
// ===== library: MasterCopy "SeachArray[FC001]" =====

FUNCTION "SeachArray[FC001]" : Void   // FC4, LAD
{ S7_Optimized_Access := 'TRUE' }
VERSION : 0.1
   VAR_INPUT
      StartSearch : Bool;
      Search : DInt;
      UserArray : Array[0..99] of Struct
         RFID : DInt;
         "Name" : String;
         ClockNumber : Int;
         AccessLevel : Int;
      END_STRUCT;
      Reset : Bool;
   END_VAR
   VAR_OUTPUT
      MatchFound : Bool;
      NoMatchFound : Bool;
      MatchIndex : Int;
      EmptyIndex : Int;
      ArrayFull : Bool;
      Done : Bool;
   END_VAR
   VAR_TEMP
      Index : Int;
      Match : Bool;
      NoMatch : Bool;
   END_VAR
   VAR CONSTANT
      Null : String;
   END_VAR
   VAR_TEMP   // added for the SCL form of the ladder/FBD networks
      _w1 : Bool;
      _w2 : Bool;
   END_VAR
BEGIN

REGION Network 1: Search For Matching RFID
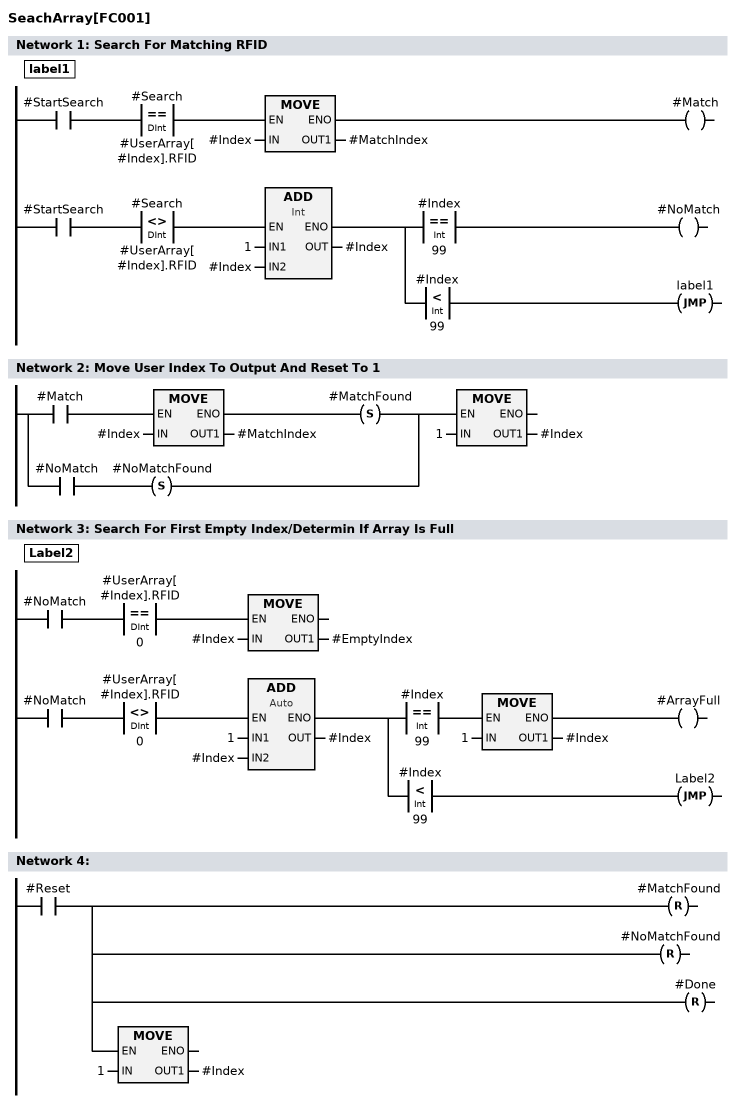
   Label( label1 )
   RUNG wire#powerrail
      Contact( #StartSearch )
      { S7_Templates := "SrcType := DInt" } EQ_Contact(in1 := #Search, in2 := #UserArray[#Index].RFID)
      Move(in := #Index, out1 => #MatchIndex)
      Coil( #Match )
   END_RUNG
   RUNG wire#powerrail
      Contact( #StartSearch )
      { S7_Templates := "SrcType := DInt" } NE_Contact(in1 := #Search, in2 := #UserArray[#Index].RFID)
      { S7_Templates := "SrcType := Int" } Add(in1 := 1, in2 := #Index, out => #Index)
      wire#w1
      { S7_Templates := "SrcType := Int" } EQ_Contact(in1 := #Index, in2 := 99)
      Coil( #NoMatch )
   END_RUNG
   RUNG wire#w1
      { S7_Templates := "SrcType := Int" } LT_Contact(in1 := #Index, in2 := 99)
      JumpCoil( label1 )
   END_RUNG
   // the same network as SCL:
   label1:
   #_w1 := #StartSearch AND (#Search = #UserArray[#Index].RFID);
   IF #_w1 THEN #MatchIndex := #Index; END_IF;
   #Match := #_w1;
   #_w2 := #StartSearch AND (#Search <> #UserArray[#Index].RFID);
   IF #_w2 THEN #Index := 1 + #Index; END_IF;
   #NoMatch := #_w2 AND (#Index = 99);
   IF #_w2 AND (#Index < 99) THEN GOTO label1; END_IF;
END_REGION

REGION Network 2: Move User Index To Output And Reset To 1
   RUNG wire#powerrail
      Contact( #Match )
      Move(in := #Index, out1 => #MatchIndex)
      S_Coil( #MatchFound )
      wire#w1
      Move(in := 1, out1 => #Index)
   END_RUNG
   RUNG wire#powerrail
      Contact( #NoMatch )
      S_Coil( #NoMatchFound )
   END_RUNG wire#w1
   // the same network as SCL:
   IF #Match THEN
       #MatchIndex := #Index;
       #MatchFound := TRUE;
   END_IF;
   IF #NoMatch THEN #NoMatchFound := TRUE; END_IF;
   IF #Match OR #NoMatch THEN #Index := 1; END_IF;
END_REGION

REGION Network 3: Search For First Empty Index/Determin If Array Is Full
   Label( Label2 )
   RUNG wire#powerrail
      Contact( #NoMatch )
      { S7_Templates := "SrcType := DInt" } EQ_Contact(in1 := #UserArray[#Index].RFID, in2 := 0)
      Move(in := #Index, out1 => #EmptyIndex)
   END_RUNG
   RUNG wire#powerrail
      Contact( #NoMatch )
      { S7_Templates := "SrcType := DInt" } NE_Contact(in1 := #UserArray[#Index].RFID, in2 := 0)
      Add(in1 := 1, in2 := #Index, out => #Index)
      wire#w1
      { S7_Templates := "SrcType := Int" } EQ_Contact(in1 := #Index, in2 := 99)
      Move(in := 1, out1 => #Index)
      Coil( #ArrayFull )
   END_RUNG
   RUNG wire#w1
      { S7_Templates := "SrcType := Int" } LT_Contact(in1 := #Index, in2 := 99)
      JumpCoil( Label2 )
   END_RUNG
   // the same network as SCL:
   Label2:
   IF #NoMatch AND (#UserArray[#Index].RFID = 0) THEN #EmptyIndex := #Index; END_IF;
   #_w1 := #NoMatch AND (#UserArray[#Index].RFID <> 0);
   IF #_w1 THEN #Index := 1 + #Index; END_IF;
   #_w2 := #_w1 AND (#Index = 99);
   IF #_w2 THEN #Index := 1; END_IF;
   #ArrayFull := #_w2;
   IF #_w1 AND (#Index < 99) THEN GOTO Label2; END_IF;
END_REGION

REGION Network 4
   RUNG wire#powerrail
      Contact( #Reset )
      wire#w1
      R_Coil( #MatchFound )
   END_RUNG
   RUNG wire#w1
      R_Coil( #NoMatchFound )
   END_RUNG
   RUNG wire#w1
      R_Coil( #Done )
   END_RUNG
   RUNG wire#w1
      Move(in := 1, out1 => #Index)
   END_RUNG
   // the same network as SCL:
   IF #Reset THEN
       #MatchFound := FALSE;
       #NoMatchFound := FALSE;
       #Done := FALSE;
       #Index := 1;
   END_IF;
END_REGION
END_FUNCTION

// ===== library: MasterCopy "LabelPrintEthernet" =====

FUNCTION "BuildLabel" : Void   // FC1, LAD
{ S7_Optimized_Access := 'TRUE' }
VERSION : 0.1
   VAR_INPUT
      REQ : Bool;
      PartNumber : String;
      PartDisctription : String;
      SerialNumber : Int;
      IPAddress1 : Byte;
      IPAddress2 : Byte;
      IPAddress3 : Byte;
      IPAddress4 : Byte;
      Port : UInt;
   END_VAR
   VAR_OUTPUT
      FinalLabel : String;
   END_VAR
   VAR_TEMP
      LabelDateTime : DTL;
      YearString : String;
      MonthString : String;
      DayString : String;
      HourString : String;
      MinuteString : String;
      SecondString : String;
      DateTimeString : String;
      AssembleLabel : String;
      SerialNumberString : String;
      BarcodeString : String;
      SerialNumberStringTemp : String;
      PrintData : String;
   END_VAR
   VAR CONSTANT
      FormatStart : String := '^XA';
      FormatLine1 : String := '^FS^A0N15,35^FO300,40^FD';
      FormatLine2 : String := '^FS^A0N20,20^FO300,80^FD';
      FormatLine3 : String := '^FS^A0N20,20^FO300,120^FD';
      FormatBarcode1 : String := '^FS^BXN,.05,200,^FO150,70^FD';
      FormatBarcode2 : String := '^FS^BXN,.04,200,^FO500,120^FD';
      FormatEnd : String := '^FS^XZ';
   END_VAR
BEGIN

REGION Network 1
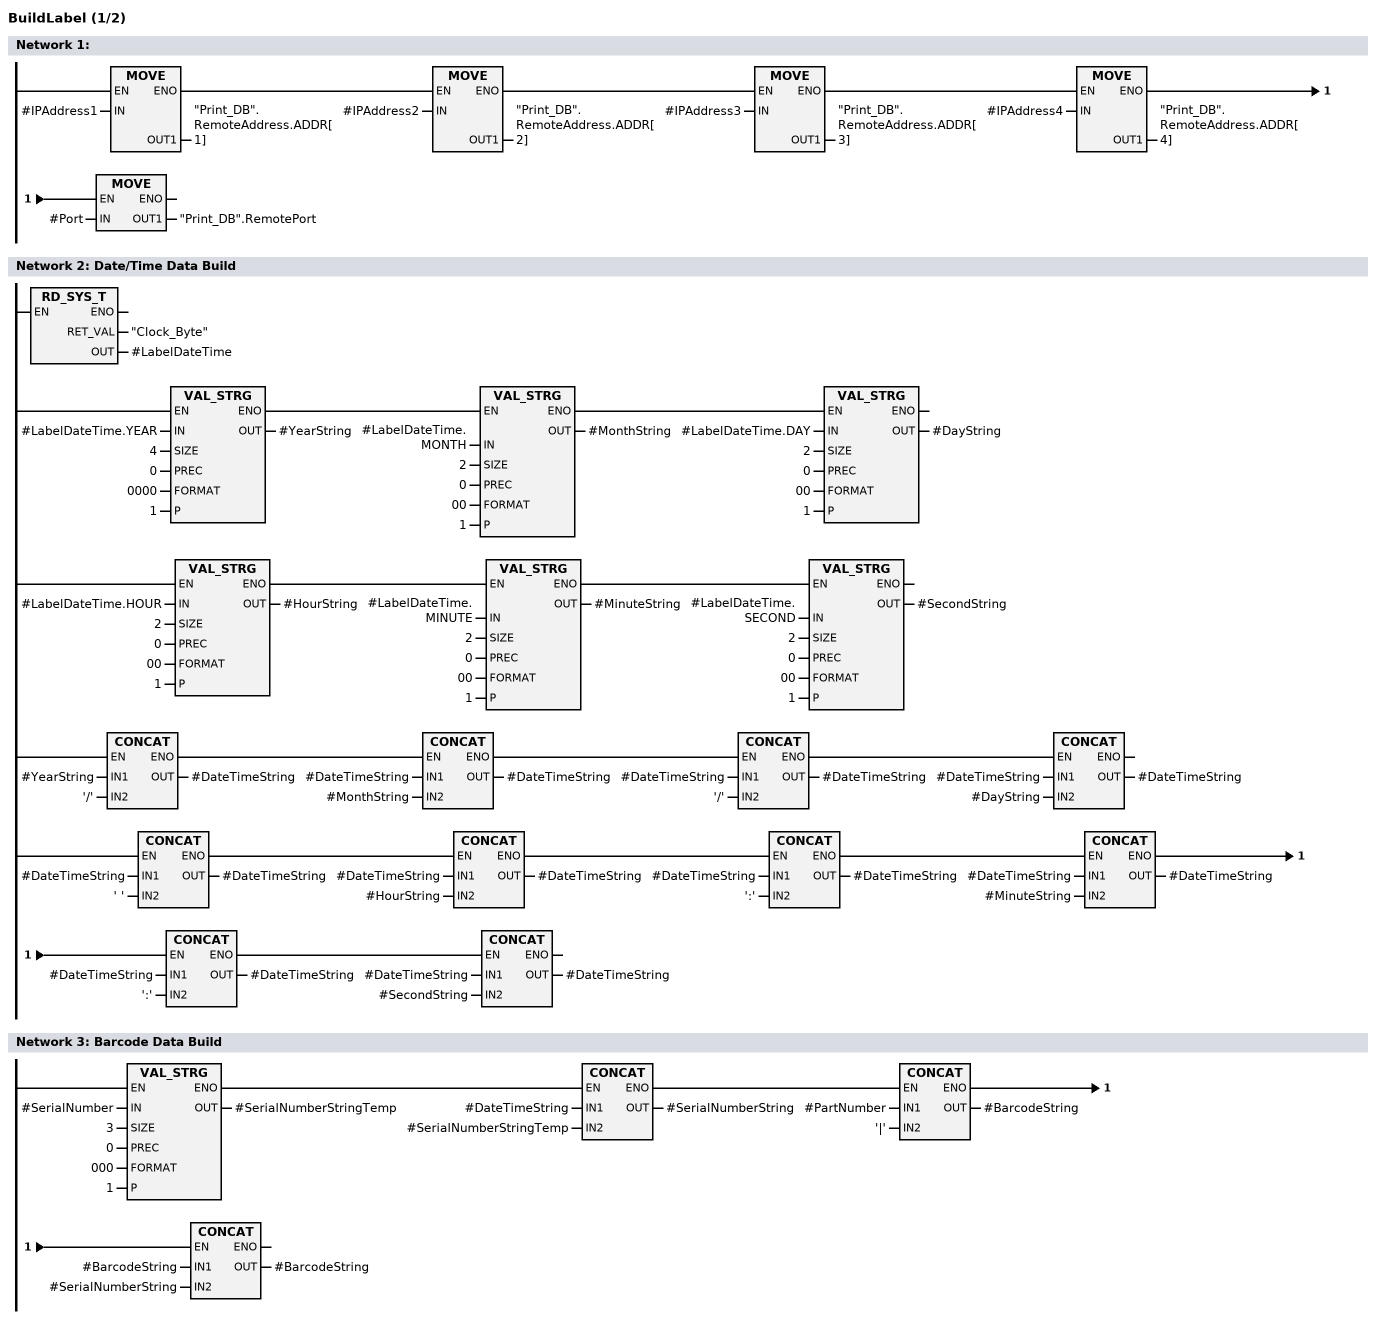
   RUNG wire#powerrail
      Move(in := #IPAddress1, out1 => "Print_DB".RemoteAddress.ADDR[1])
      Move(in := #IPAddress2, out1 => "Print_DB".RemoteAddress.ADDR[2])
      Move(in := #IPAddress3, out1 => "Print_DB".RemoteAddress.ADDR[3])
      Move(in := #IPAddress4, out1 => "Print_DB".RemoteAddress.ADDR[4])
      Move(in := #Port, out1 => "Print_DB".RemotePort)
   END_RUNG
   // the same network as SCL:
   "Print_DB".RemoteAddress.ADDR[1] := #IPAddress1;
   "Print_DB".RemoteAddress.ADDR[2] := #IPAddress2;
   "Print_DB".RemoteAddress.ADDR[3] := #IPAddress3;
   "Print_DB".RemoteAddress.ADDR[4] := #IPAddress4;
   "Print_DB".RemotePort := #Port;
END_REGION

REGION Network 2: Date/Time Data Build
   // ENO of a box is taken as its EN; it also drops when the box reports an error
   "Clock_Byte" := RD_SYS_T(OUT => #LabelDateTime);
   VAL_STRG(IN := #LabelDateTime.YEAR, SIZE := 4, PREC := 0, FORMAT := 0000, P := 1, OUT => #YearString);
   VAL_STRG(IN := #LabelDateTime.MONTH, SIZE := 2, PREC := 0, FORMAT := 00, P := 1, OUT => #MonthString);
   VAL_STRG(IN := #LabelDateTime.DAY, SIZE := 2, PREC := 0, FORMAT := 00, P := 1, OUT => #DayString);
   VAL_STRG(IN := #LabelDateTime.HOUR, SIZE := 2, PREC := 0, FORMAT := 00, P := 1, OUT => #HourString);
   VAL_STRG(IN := #LabelDateTime.MINUTE, SIZE := 2, PREC := 0, FORMAT := 00, P := 1, OUT => #MinuteString);
   VAL_STRG(IN := #LabelDateTime.SECOND, SIZE := 2, PREC := 0, FORMAT := 00, P := 1, OUT => #SecondString);
   #DateTimeString := CONCAT(IN1 := #YearString, IN2 := '/');
   #DateTimeString := CONCAT(IN1 := #DateTimeString, IN2 := #MonthString);
   #DateTimeString := CONCAT(IN1 := #DateTimeString, IN2 := '/');
   #DateTimeString := CONCAT(IN1 := #DateTimeString, IN2 := #DayString);
   #DateTimeString := CONCAT(IN1 := #DateTimeString, IN2 := ' ');
   #DateTimeString := CONCAT(IN1 := #DateTimeString, IN2 := #HourString);
   #DateTimeString := CONCAT(IN1 := #DateTimeString, IN2 := ':');
   #DateTimeString := CONCAT(IN1 := #DateTimeString, IN2 := #MinuteString);
   #DateTimeString := CONCAT(IN1 := #DateTimeString, IN2 := ':');
   #DateTimeString := CONCAT(IN1 := #DateTimeString, IN2 := #SecondString);
END_REGION

REGION Network 3: Barcode Data Build
   // ENO of a box is taken as its EN; it also drops when the box reports an error
   VAL_STRG(IN := #SerialNumber, SIZE := 3, PREC := 0, FORMAT := 000, P := 1, OUT => #SerialNumberStringTemp);
   #SerialNumberString := CONCAT(IN1 := #DateTimeString, IN2 := #SerialNumberStringTemp);
   #BarcodeString := CONCAT(IN1 := #PartNumber, IN2 := '|');
   #BarcodeString := CONCAT(IN1 := #BarcodeString, IN2 := #SerialNumberString);
END_REGION

REGION Network 4: Label Data Build
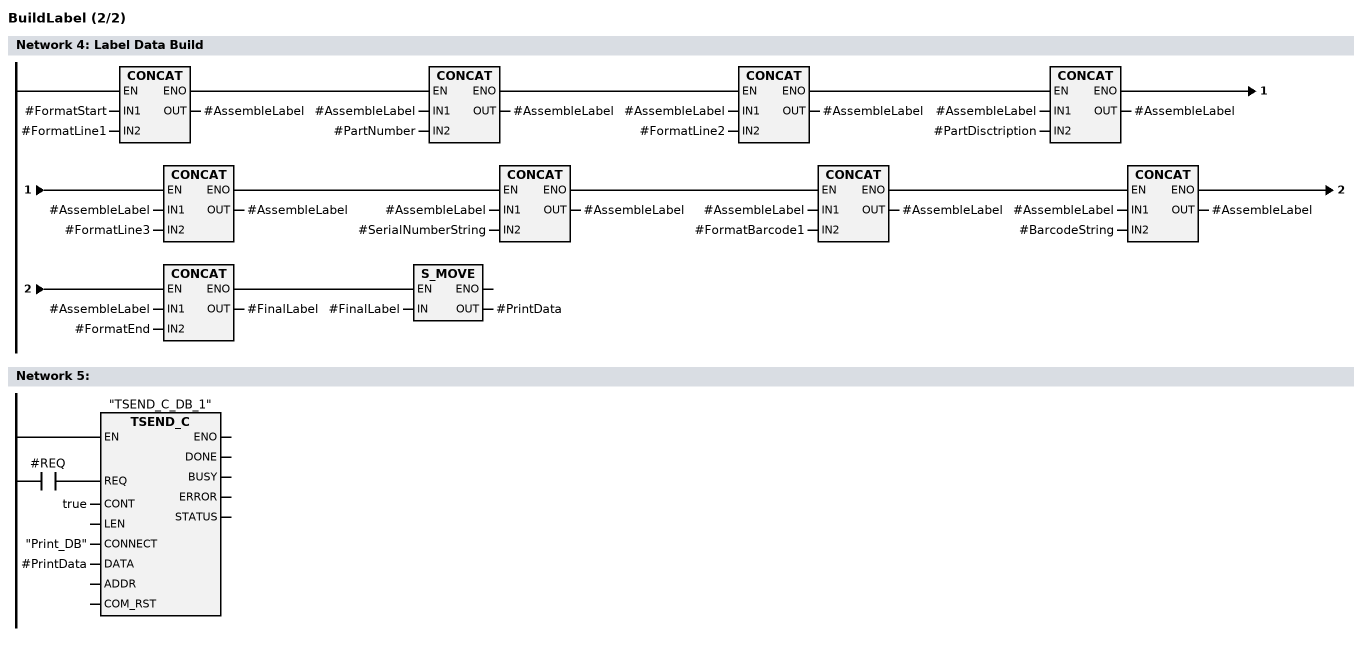
   #AssembleLabel := CONCAT(IN1 := #FormatStart, IN2 := #FormatLine1);
   #AssembleLabel := CONCAT(IN1 := #AssembleLabel, IN2 := #PartNumber);
   #AssembleLabel := CONCAT(IN1 := #AssembleLabel, IN2 := #FormatLine2);
   #AssembleLabel := CONCAT(IN1 := #AssembleLabel, IN2 := #PartDisctription);
   #AssembleLabel := CONCAT(IN1 := #AssembleLabel, IN2 := #FormatLine3);
   #AssembleLabel := CONCAT(IN1 := #AssembleLabel, IN2 := #SerialNumberString);
   #AssembleLabel := CONCAT(IN1 := #AssembleLabel, IN2 := #FormatBarcode1);
   #AssembleLabel := CONCAT(IN1 := #AssembleLabel, IN2 := #BarcodeString);
   #FinalLabel := CONCAT(IN1 := #AssembleLabel, IN2 := #FormatEnd);
   #PrintData := #FinalLabel;
END_REGION

REGION Network 5
   "TSEND_C_DB_1"(REQ := #REQ, CONT := true, CONNECT := "Print_DB", DATA := #PrintData);   // TSEND_C
END_REGION
END_FUNCTION

// ===== library: MasterCopy "Banner_IOLink_K50L" =====

FUNCTION "Banner_IOLink_K50L" : Void   // FC6, LAD
{ S7_Optimized_Access := 'TRUE' }
VERSION : 0.1
   VAR_INPUT
      IN : Bool;
      "Color 1" : Int;
      "Color 1 Intensity" : Int;
      "Color 2" : Int;
      "Color 2 Intensity" : Int;
      "Animation Type" : Int;
      "Rotation Direction" : Bool;
      "Flash Rate" : Int;
   END_VAR
BEGIN

REGION Network 1
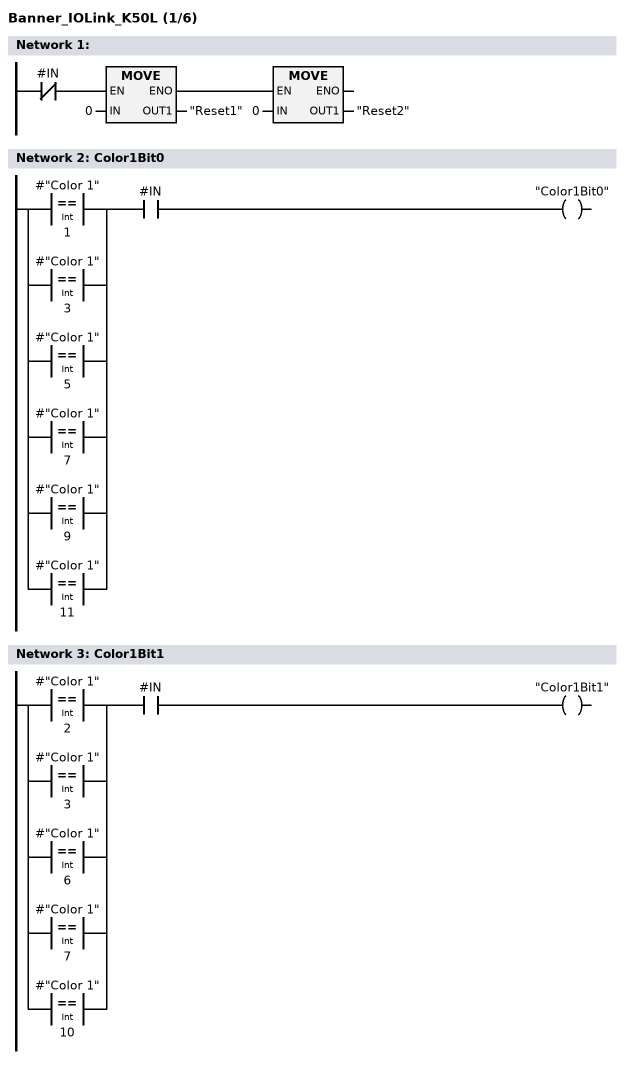
   RUNG wire#powerrail
      I_Contact( #IN )
      Move(in := 0, out1 => "Reset1")
      Move(in := 0, out1 => "Reset2")
   END_RUNG
   // the same network as SCL:
   IF NOT #IN THEN
       "Reset1" := 0;
       "Reset2" := 0;
   END_IF;
END_REGION

REGION Network 2: Color1Bit0
   RUNG wire#powerrail
      { S7_Templates := "SrcType := Int" } EQ_Contact(in1 := #"Color 1", in2 := 1)
      wire#w1
      Contact( #IN )
      Coil( "Color1Bit0" )
   END_RUNG
   RUNG wire#powerrail
      { S7_Templates := "SrcType := Int" } EQ_Contact(in1 := #"Color 1", in2 := 3)
   END_RUNG wire#w1
   RUNG wire#powerrail
      { S7_Templates := "SrcType := Int" } EQ_Contact(in1 := #"Color 1", in2 := 5)
   END_RUNG wire#w1
   RUNG wire#powerrail
      { S7_Templates := "SrcType := Int" } EQ_Contact(in1 := #"Color 1", in2 := 7)
   END_RUNG wire#w1
   RUNG wire#powerrail
      { S7_Templates := "SrcType := Int" } EQ_Contact(in1 := #"Color 1", in2 := 9)
   END_RUNG wire#w1
   RUNG wire#powerrail
      { S7_Templates := "SrcType := Int" } EQ_Contact(in1 := #"Color 1", in2 := 11)
   END_RUNG wire#w1
   // the same network as SCL:
   "Color1Bit0" := ((#"Color 1" = 1) OR (#"Color 1" = 3) OR (#"Color 1" = 5) OR (#"Color 1" = 7) OR (#"Color 1" = 9) OR (#"Color 1" = 11)) AND #IN;
END_REGION

REGION Network 3: Color1Bit1
   RUNG wire#powerrail
      { S7_Templates := "SrcType := Int" } EQ_Contact(in1 := #"Color 1", in2 := 2)
      wire#w1
      Contact( #IN )
      Coil( "Color1Bit1" )
   END_RUNG
   RUNG wire#powerrail
      { S7_Templates := "SrcType := Int" } EQ_Contact(in1 := #"Color 1", in2 := 3)
   END_RUNG wire#w1
   RUNG wire#powerrail
      { S7_Templates := "SrcType := Int" } EQ_Contact(in1 := #"Color 1", in2 := 6)
   END_RUNG wire#w1
   RUNG wire#powerrail
      { S7_Templates := "SrcType := Int" } EQ_Contact(in1 := #"Color 1", in2 := 7)
   END_RUNG wire#w1
   RUNG wire#powerrail
      { S7_Templates := "SrcType := Int" } EQ_Contact(in1 := #"Color 1", in2 := 10)
   END_RUNG wire#w1
   // the same network as SCL:
   "Color1Bit1" := ((#"Color 1" = 2) OR (#"Color 1" = 3) OR (#"Color 1" = 6) OR (#"Color 1" = 7) OR (#"Color 1" = 10)) AND #IN;
END_REGION

REGION Network 4: Color1Bit2
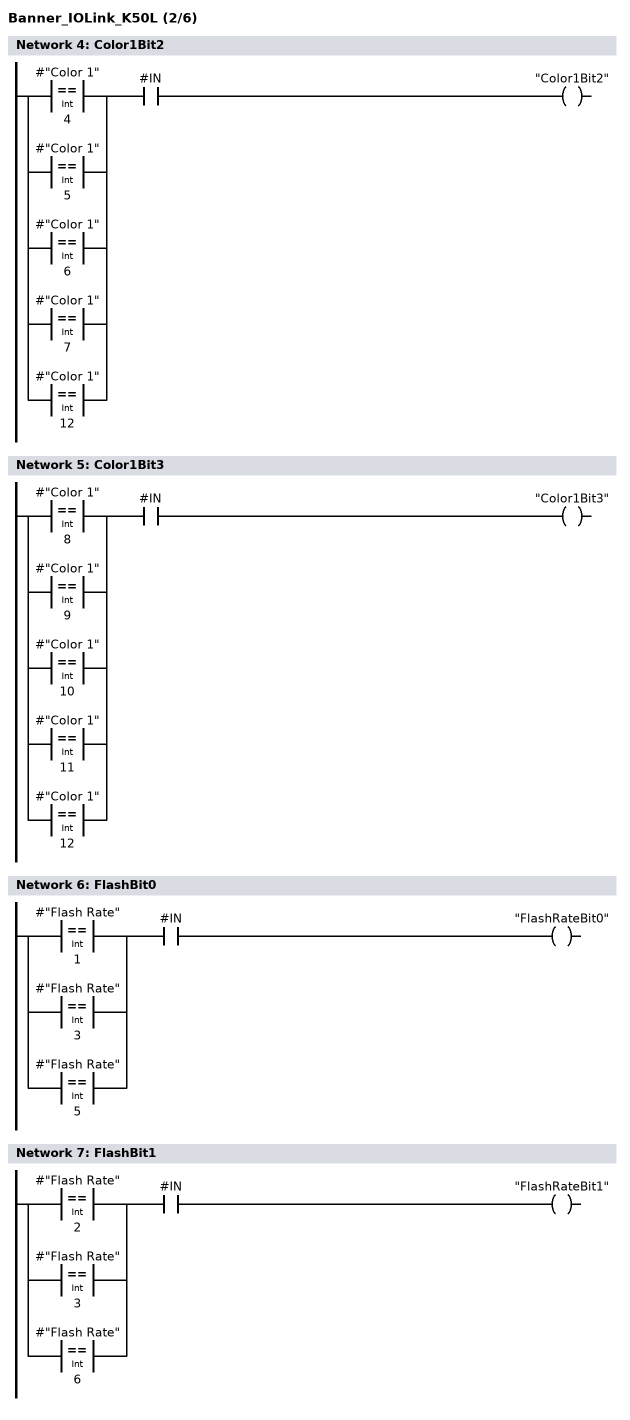
   RUNG wire#powerrail
      { S7_Templates := "SrcType := Int" } EQ_Contact(in1 := #"Color 1", in2 := 4)
      wire#w1
      Contact( #IN )
      Coil( "Color1Bit2" )
   END_RUNG
   RUNG wire#powerrail
      { S7_Templates := "SrcType := Int" } EQ_Contact(in1 := #"Color 1", in2 := 5)
   END_RUNG wire#w1
   RUNG wire#powerrail
      { S7_Templates := "SrcType := Int" } EQ_Contact(in1 := #"Color 1", in2 := 6)
   END_RUNG wire#w1
   RUNG wire#powerrail
      { S7_Templates := "SrcType := Int" } EQ_Contact(in1 := #"Color 1", in2 := 7)
   END_RUNG wire#w1
   RUNG wire#powerrail
      { S7_Templates := "SrcType := Int" } EQ_Contact(in1 := #"Color 1", in2 := 12)
   END_RUNG wire#w1
   // the same network as SCL:
   "Color1Bit2" := ((#"Color 1" = 4) OR (#"Color 1" = 5) OR (#"Color 1" = 6) OR (#"Color 1" = 7) OR (#"Color 1" = 12)) AND #IN;
END_REGION

REGION Network 5: Color1Bit3
   RUNG wire#powerrail
      { S7_Templates := "SrcType := Int" } EQ_Contact(in1 := #"Color 1", in2 := 8)
      wire#w1
      Contact( #IN )
      Coil( "Color1Bit3" )
   END_RUNG
   RUNG wire#powerrail
      { S7_Templates := "SrcType := Int" } EQ_Contact(in1 := #"Color 1", in2 := 9)
   END_RUNG wire#w1
   RUNG wire#powerrail
      { S7_Templates := "SrcType := Int" } EQ_Contact(in1 := #"Color 1", in2 := 10)
   END_RUNG wire#w1
   RUNG wire#powerrail
      { S7_Templates := "SrcType := Int" } EQ_Contact(in1 := #"Color 1", in2 := 11)
   END_RUNG wire#w1
   RUNG wire#powerrail
      { S7_Templates := "SrcType := Int" } EQ_Contact(in1 := #"Color 1", in2 := 12)
   END_RUNG wire#w1
   // the same network as SCL:
   "Color1Bit3" := ((#"Color 1" = 8) OR (#"Color 1" = 9) OR (#"Color 1" = 10) OR (#"Color 1" = 11) OR (#"Color 1" = 12)) AND #IN;
END_REGION

REGION Network 6: FlashBit0
   RUNG wire#powerrail
      { S7_Templates := "SrcType := Int" } EQ_Contact(in1 := #"Flash Rate", in2 := 1)
      wire#w1
      Contact( #IN )
      Coil( "FlashRateBit0" )
   END_RUNG
   RUNG wire#powerrail
      { S7_Templates := "SrcType := Int" } EQ_Contact(in1 := #"Flash Rate", in2 := 3)
   END_RUNG wire#w1
   RUNG wire#powerrail
      { S7_Templates := "SrcType := Int" } EQ_Contact(in1 := #"Flash Rate", in2 := 5)
   END_RUNG wire#w1
   // the same network as SCL:
   "FlashRateBit0" := ((#"Flash Rate" = 1) OR (#"Flash Rate" = 3) OR (#"Flash Rate" = 5)) AND #IN;
END_REGION

REGION Network 7: FlashBit1
   RUNG wire#powerrail
      { S7_Templates := "SrcType := Int" } EQ_Contact(in1 := #"Flash Rate", in2 := 2)
      wire#w1
      Contact( #IN )
      Coil( "FlashRateBit1" )
   END_RUNG
   RUNG wire#powerrail
      { S7_Templates := "SrcType := Int" } EQ_Contact(in1 := #"Flash Rate", in2 := 3)
   END_RUNG wire#w1
   RUNG wire#powerrail
      { S7_Templates := "SrcType := Int" } EQ_Contact(in1 := #"Flash Rate", in2 := 6)
   END_RUNG wire#w1
   // the same network as SCL:
   "FlashRateBit1" := ((#"Flash Rate" = 2) OR (#"Flash Rate" = 3) OR (#"Flash Rate" = 6)) AND #IN;
END_REGION

REGION Network 8: FlashBit2
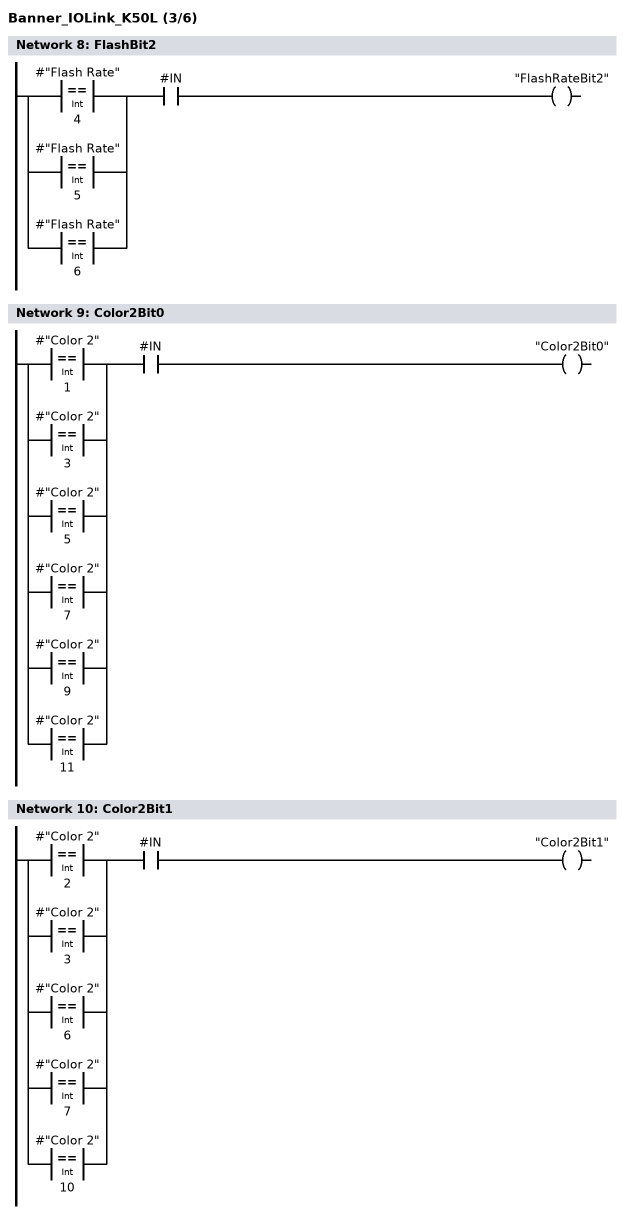
   RUNG wire#powerrail
      { S7_Templates := "SrcType := Int" } EQ_Contact(in1 := #"Flash Rate", in2 := 4)
      wire#w1
      Contact( #IN )
      Coil( "FlashRateBit2" )
   END_RUNG
   RUNG wire#powerrail
      { S7_Templates := "SrcType := Int" } EQ_Contact(in1 := #"Flash Rate", in2 := 5)
   END_RUNG wire#w1
   RUNG wire#powerrail
      { S7_Templates := "SrcType := Int" } EQ_Contact(in1 := #"Flash Rate", in2 := 6)
   END_RUNG wire#w1
   // the same network as SCL:
   "FlashRateBit2" := ((#"Flash Rate" = 4) OR (#"Flash Rate" = 5) OR (#"Flash Rate" = 6)) AND #IN;
END_REGION

REGION Network 9: Color2Bit0
   RUNG wire#powerrail
      { S7_Templates := "SrcType := Int" } EQ_Contact(in1 := #"Color 2", in2 := 1)
      wire#w1
      Contact( #IN )
      Coil( "Color2Bit0" )
   END_RUNG
   RUNG wire#powerrail
      { S7_Templates := "SrcType := Int" } EQ_Contact(in1 := #"Color 2", in2 := 3)
   END_RUNG wire#w1
   RUNG wire#powerrail
      { S7_Templates := "SrcType := Int" } EQ_Contact(in1 := #"Color 2", in2 := 5)
   END_RUNG wire#w1
   RUNG wire#powerrail
      { S7_Templates := "SrcType := Int" } EQ_Contact(in1 := #"Color 2", in2 := 7)
   END_RUNG wire#w1
   RUNG wire#powerrail
      { S7_Templates := "SrcType := Int" } EQ_Contact(in1 := #"Color 2", in2 := 9)
   END_RUNG wire#w1
   RUNG wire#powerrail
      { S7_Templates := "SrcType := Int" } EQ_Contact(in1 := #"Color 2", in2 := 11)
   END_RUNG wire#w1
   // the same network as SCL:
   "Color2Bit0" := ((#"Color 2" = 1) OR (#"Color 2" = 3) OR (#"Color 2" = 5) OR (#"Color 2" = 7) OR (#"Color 2" = 9) OR (#"Color 2" = 11)) AND #IN;
END_REGION

REGION Network 10: Color2Bit1
   RUNG wire#powerrail
      { S7_Templates := "SrcType := Int" } EQ_Contact(in1 := #"Color 2", in2 := 2)
      wire#w1
      Contact( #IN )
      Coil( "Color2Bit1" )
   END_RUNG
   RUNG wire#powerrail
      { S7_Templates := "SrcType := Int" } EQ_Contact(in1 := #"Color 2", in2 := 3)
   END_RUNG wire#w1
   RUNG wire#powerrail
      { S7_Templates := "SrcType := Int" } EQ_Contact(in1 := #"Color 2", in2 := 6)
   END_RUNG wire#w1
   RUNG wire#powerrail
      { S7_Templates := "SrcType := Int" } EQ_Contact(in1 := #"Color 2", in2 := 7)
   END_RUNG wire#w1
   RUNG wire#powerrail
      { S7_Templates := "SrcType := Int" } EQ_Contact(in1 := #"Color 2", in2 := 10)
   END_RUNG wire#w1
   // the same network as SCL:
   "Color2Bit1" := ((#"Color 2" = 2) OR (#"Color 2" = 3) OR (#"Color 2" = 6) OR (#"Color 2" = 7) OR (#"Color 2" = 10)) AND #IN;
END_REGION

REGION Network 11: Color2Bit2
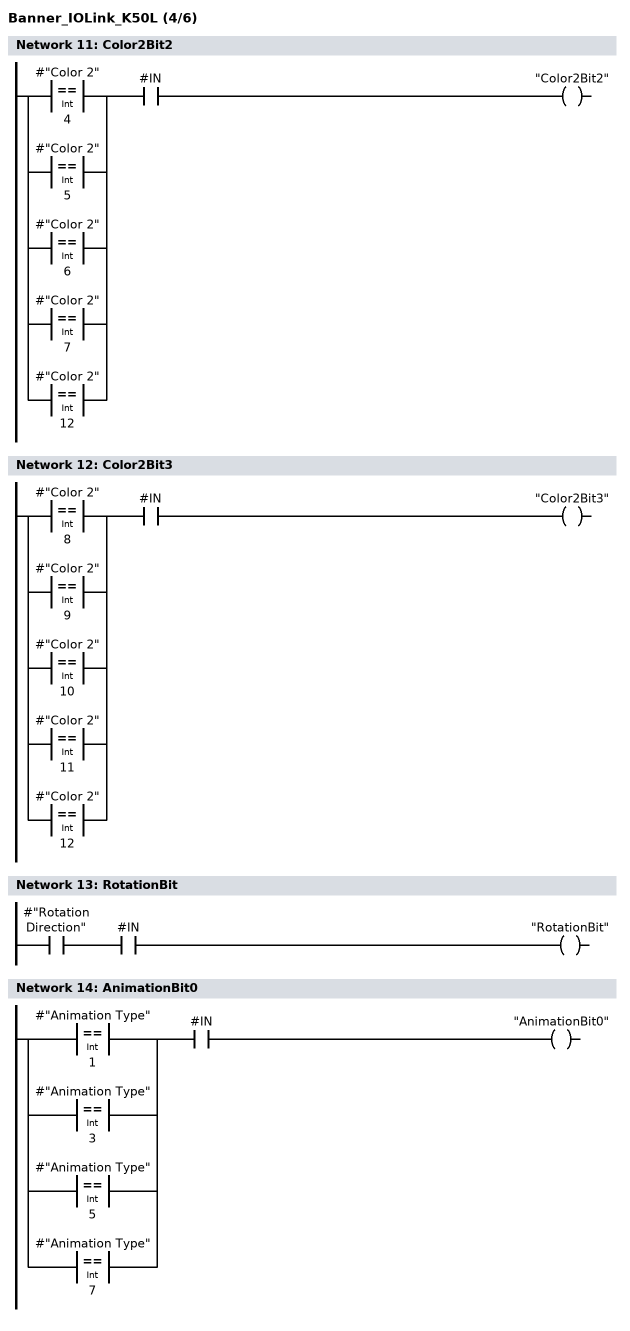
   RUNG wire#powerrail
      { S7_Templates := "SrcType := Int" } EQ_Contact(in1 := #"Color 2", in2 := 4)
      wire#w1
      Contact( #IN )
      Coil( "Color2Bit2" )
   END_RUNG
   RUNG wire#powerrail
      { S7_Templates := "SrcType := Int" } EQ_Contact(in1 := #"Color 2", in2 := 5)
   END_RUNG wire#w1
   RUNG wire#powerrail
      { S7_Templates := "SrcType := Int" } EQ_Contact(in1 := #"Color 2", in2 := 6)
   END_RUNG wire#w1
   RUNG wire#powerrail
      { S7_Templates := "SrcType := Int" } EQ_Contact(in1 := #"Color 2", in2 := 7)
   END_RUNG wire#w1
   RUNG wire#powerrail
      { S7_Templates := "SrcType := Int" } EQ_Contact(in1 := #"Color 2", in2 := 12)
   END_RUNG wire#w1
   // the same network as SCL:
   "Color2Bit2" := ((#"Color 2" = 4) OR (#"Color 2" = 5) OR (#"Color 2" = 6) OR (#"Color 2" = 7) OR (#"Color 2" = 12)) AND #IN;
END_REGION

REGION Network 12: Color2Bit3
   RUNG wire#powerrail
      { S7_Templates := "SrcType := Int" } EQ_Contact(in1 := #"Color 2", in2 := 8)
      wire#w1
      Contact( #IN )
      Coil( "Color2Bit3" )
   END_RUNG
   RUNG wire#powerrail
      { S7_Templates := "SrcType := Int" } EQ_Contact(in1 := #"Color 2", in2 := 9)
   END_RUNG wire#w1
   RUNG wire#powerrail
      { S7_Templates := "SrcType := Int" } EQ_Contact(in1 := #"Color 2", in2 := 10)
   END_RUNG wire#w1
   RUNG wire#powerrail
      { S7_Templates := "SrcType := Int" } EQ_Contact(in1 := #"Color 2", in2 := 11)
   END_RUNG wire#w1
   RUNG wire#powerrail
      { S7_Templates := "SrcType := Int" } EQ_Contact(in1 := #"Color 2", in2 := 12)
   END_RUNG wire#w1
   // the same network as SCL:
   "Color2Bit3" := ((#"Color 2" = 8) OR (#"Color 2" = 9) OR (#"Color 2" = 10) OR (#"Color 2" = 11) OR (#"Color 2" = 12)) AND #IN;
END_REGION

REGION Network 13: RotationBit
   RUNG wire#powerrail
      Contact( #"Rotation Direction" )
      Contact( #IN )
      Coil( "RotationBit" )
   END_RUNG
   // the same network as SCL:
   "RotationBit" := #"Rotation Direction" AND #IN;
END_REGION

REGION Network 14: AnimationBit0
   RUNG wire#powerrail
      { S7_Templates := "SrcType := Int" } EQ_Contact(in1 := #"Animation Type", in2 := 1)
      wire#w1
      Contact( #IN )
      Coil( "AnimationBit0" )
   END_RUNG
   RUNG wire#powerrail
      { S7_Templates := "SrcType := Int" } EQ_Contact(in1 := #"Animation Type", in2 := 3)
   END_RUNG wire#w1
   RUNG wire#powerrail
      { S7_Templates := "SrcType := Int" } EQ_Contact(in1 := #"Animation Type", in2 := 5)
   END_RUNG wire#w1
   RUNG wire#powerrail
      { S7_Templates := "SrcType := Int" } EQ_Contact(in1 := #"Animation Type", in2 := 7)
   END_RUNG wire#w1
   // the same network as SCL:
   "AnimationBit0" := ((#"Animation Type" = 1) OR (#"Animation Type" = 3) OR (#"Animation Type" = 5) OR (#"Animation Type" = 7)) AND #IN;
END_REGION

REGION Network 15: AnimationBit1
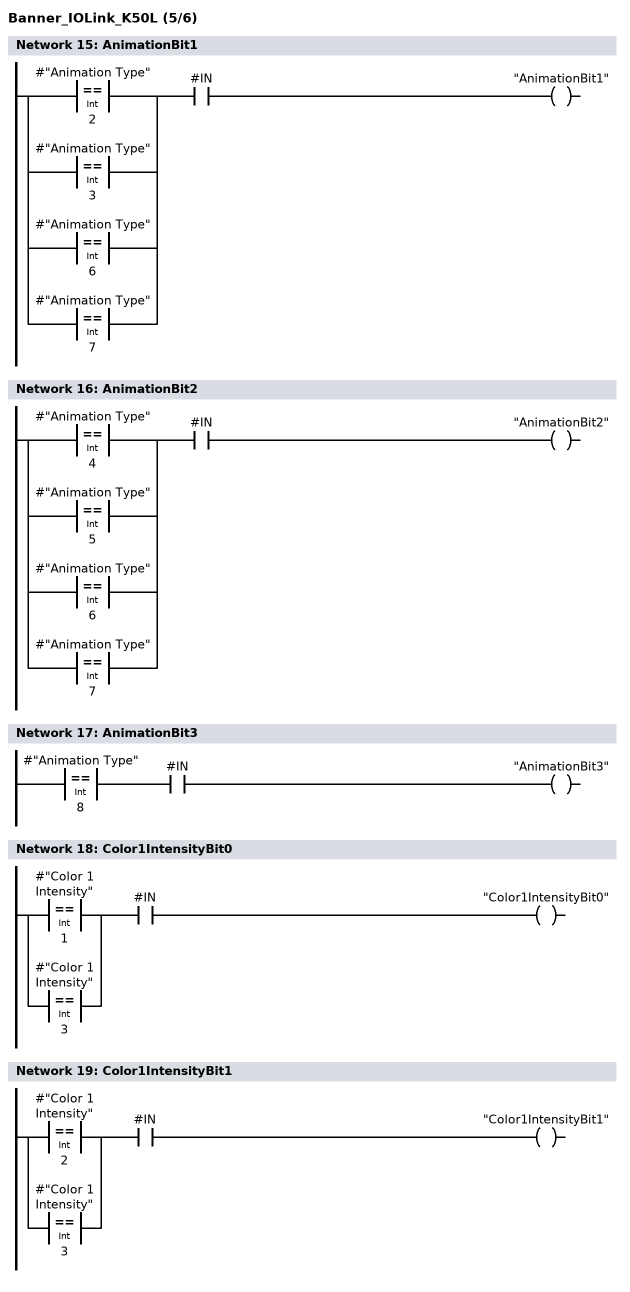
   RUNG wire#powerrail
      { S7_Templates := "SrcType := Int" } EQ_Contact(in1 := #"Animation Type", in2 := 2)
      wire#w1
      Contact( #IN )
      Coil( "AnimationBit1" )
   END_RUNG
   RUNG wire#powerrail
      { S7_Templates := "SrcType := Int" } EQ_Contact(in1 := #"Animation Type", in2 := 3)
   END_RUNG wire#w1
   RUNG wire#powerrail
      { S7_Templates := "SrcType := Int" } EQ_Contact(in1 := #"Animation Type", in2 := 6)
   END_RUNG wire#w1
   RUNG wire#powerrail
      { S7_Templates := "SrcType := Int" } EQ_Contact(in1 := #"Animation Type", in2 := 7)
   END_RUNG wire#w1
   // the same network as SCL:
   "AnimationBit1" := ((#"Animation Type" = 2) OR (#"Animation Type" = 3) OR (#"Animation Type" = 6) OR (#"Animation Type" = 7)) AND #IN;
END_REGION

REGION Network 16: AnimationBit2
   RUNG wire#powerrail
      { S7_Templates := "SrcType := Int" } EQ_Contact(in1 := #"Animation Type", in2 := 4)
      wire#w1
      Contact( #IN )
      Coil( "AnimationBit2" )
   END_RUNG
   RUNG wire#powerrail
      { S7_Templates := "SrcType := Int" } EQ_Contact(in1 := #"Animation Type", in2 := 5)
   END_RUNG wire#w1
   RUNG wire#powerrail
      { S7_Templates := "SrcType := Int" } EQ_Contact(in1 := #"Animation Type", in2 := 6)
   END_RUNG wire#w1
   RUNG wire#powerrail
      { S7_Templates := "SrcType := Int" } EQ_Contact(in1 := #"Animation Type", in2 := 7)
   END_RUNG wire#w1
   // the same network as SCL:
   "AnimationBit2" := ((#"Animation Type" = 4) OR (#"Animation Type" = 5) OR (#"Animation Type" = 6) OR (#"Animation Type" = 7)) AND #IN;
END_REGION

REGION Network 17: AnimationBit3
   RUNG wire#powerrail
      { S7_Templates := "SrcType := Int" } EQ_Contact(in1 := #"Animation Type", in2 := 8)
      Contact( #IN )
      Coil( "AnimationBit3" )
   END_RUNG
   // the same network as SCL:
   "AnimationBit3" := (#"Animation Type" = 8) AND #IN;
END_REGION

REGION Network 18: Color1IntensityBit0
   RUNG wire#powerrail
      { S7_Templates := "SrcType := Int" } EQ_Contact(in1 := #"Color 1 Intensity", in2 := 1)
      wire#w1
      Contact( #IN )
      Coil( "Color1IntensityBit0" )
   END_RUNG
   RUNG wire#powerrail
      { S7_Templates := "SrcType := Int" } EQ_Contact(in1 := #"Color 1 Intensity", in2 := 3)
   END_RUNG wire#w1
   // the same network as SCL:
   "Color1IntensityBit0" := ((#"Color 1 Intensity" = 1) OR (#"Color 1 Intensity" = 3)) AND #IN;
END_REGION

REGION Network 19: Color1IntensityBit1
   RUNG wire#powerrail
      { S7_Templates := "SrcType := Int" } EQ_Contact(in1 := #"Color 1 Intensity", in2 := 2)
      wire#w1
      Contact( #IN )
      Coil( "Color1IntensityBit1" )
   END_RUNG
   RUNG wire#powerrail
      { S7_Templates := "SrcType := Int" } EQ_Contact(in1 := #"Color 1 Intensity", in2 := 3)
   END_RUNG wire#w1
   // the same network as SCL:
   "Color1IntensityBit1" := ((#"Color 1 Intensity" = 2) OR (#"Color 1 Intensity" = 3)) AND #IN;
END_REGION

REGION Network 20: Color1IntensityBit2
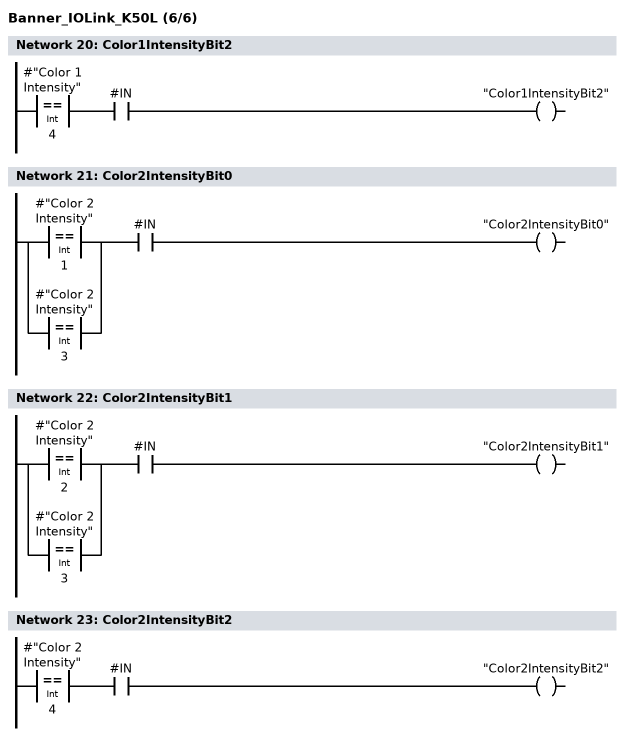
   RUNG wire#powerrail
      { S7_Templates := "SrcType := Int" } EQ_Contact(in1 := #"Color 1 Intensity", in2 := 4)
      Contact( #IN )
      Coil( "Color1IntensityBit2" )
   END_RUNG
   // the same network as SCL:
   "Color1IntensityBit2" := (#"Color 1 Intensity" = 4) AND #IN;
END_REGION

REGION Network 21: Color2IntensityBit0
   RUNG wire#powerrail
      { S7_Templates := "SrcType := Int" } EQ_Contact(in1 := #"Color 2 Intensity", in2 := 1)
      wire#w1
      Contact( #IN )
      Coil( "Color2IntensityBit0" )
   END_RUNG
   RUNG wire#powerrail
      { S7_Templates := "SrcType := Int" } EQ_Contact(in1 := #"Color 2 Intensity", in2 := 3)
   END_RUNG wire#w1
   // the same network as SCL:
   "Color2IntensityBit0" := ((#"Color 2 Intensity" = 1) OR (#"Color 2 Intensity" = 3)) AND #IN;
END_REGION

REGION Network 22: Color2IntensityBit1
   RUNG wire#powerrail
      { S7_Templates := "SrcType := Int" } EQ_Contact(in1 := #"Color 2 Intensity", in2 := 2)
      wire#w1
      Contact( #IN )
      Coil( "Color2IntensityBit1" )
   END_RUNG
   RUNG wire#powerrail
      { S7_Templates := "SrcType := Int" } EQ_Contact(in1 := #"Color 2 Intensity", in2 := 3)
   END_RUNG wire#w1
   // the same network as SCL:
   "Color2IntensityBit1" := ((#"Color 2 Intensity" = 2) OR (#"Color 2 Intensity" = 3)) AND #IN;
END_REGION

REGION Network 23: Color2IntensityBit2
   RUNG wire#powerrail
      { S7_Templates := "SrcType := Int" } EQ_Contact(in1 := #"Color 2 Intensity", in2 := 4)
      Contact( #IN )
      Coil( "Color2IntensityBit2" )
   END_RUNG
   // the same network as SCL:
   "Color2IntensityBit2" := (#"Color 2 Intensity" = 4) AND #IN;
END_REGION
END_FUNCTION

// ===== library: MasterCopy "LabelPrintRS232" =====

FUNCTION_BLOCK "PrintLabel"   // FB1, LAD
{ S7_Optimized_Access := 'TRUE' }
VERSION : 0.1
   VAR_INPUT
      Print : Bool;
      PartNumber : String;
      PartDisctription : String;
      SerialNumber : Int;
      Port : Port;
   END_VAR
   VAR_TEMP
      LabelDateTime : DTL;
      YearString : String;
      MonthString : String;
      DayString : String;
      SecondString : String;
      MinuteString : String;
      HourString : String;
      DateTimeString : String;
      SerialNumberStringTemp : String;
      SerialNumberString : String;
      BarcodeString : String;
      Line1String : String;
      Enable : Bool;
      Line1Done : Bool;
      Line1Error : Bool;
      Line1Status : Word;
      Line2String : String;
      Line2Done : Bool;
      Line2Error : Bool;
      Line2Status : Word;
      Line3String : String;
      Line3Done : Bool;
      Line3Error : Bool;
      Line3Status : Word;
      BarcodeStringTemp : String;
      BarcodeDone : Bool;
      BarcodeError : Bool;
      BarcodeStatus : Word;
   END_VAR
   VAR CONSTANT
      FormatStart : String := '^XA~SD25^PW900';
      FormatLine1 : String := '^FS^A0N15,35^FO300,40^FD';
      FormatLine2 : String := '^FS^A0N15,25^FO300,80^FD';
      FormatLine3 : String := '^FS^A0N15,25^FO300,110^FD';
      FormatBarcode1 : String := '^FS^BXN,.05,200^FH,50,N^FO150,40^FD';
      FormatEnd : String := '^FS^XZ';
   END_VAR
BEGIN

REGION Network 2: Date/Time Data Build
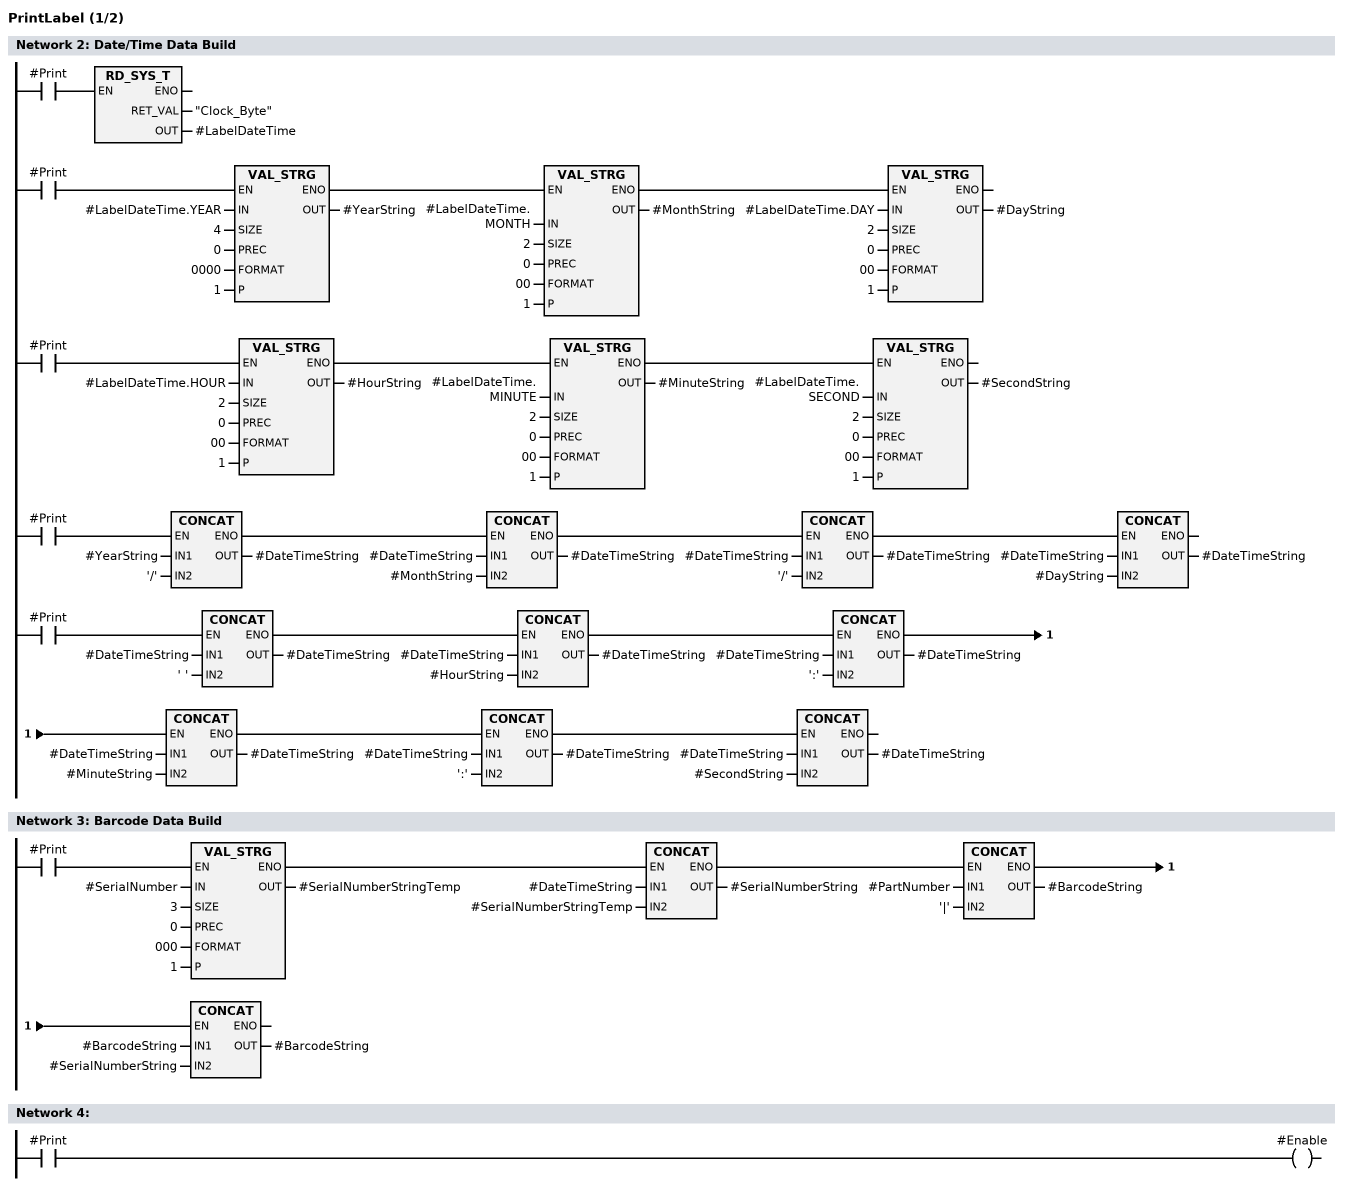
   // ENO of a box is taken as its EN; it also drops when the box reports an error
   IF #Print THEN
       "Clock_Byte" := RD_SYS_T(OUT => #LabelDateTime);
       VAL_STRG(IN := #LabelDateTime.YEAR, SIZE := 4, PREC := 0, FORMAT := 0000, P := 1, OUT => #YearString);
       VAL_STRG(IN := #LabelDateTime.MONTH, SIZE := 2, PREC := 0, FORMAT := 00, P := 1, OUT => #MonthString);
       VAL_STRG(IN := #LabelDateTime.DAY, SIZE := 2, PREC := 0, FORMAT := 00, P := 1, OUT => #DayString);
       VAL_STRG(IN := #LabelDateTime.HOUR, SIZE := 2, PREC := 0, FORMAT := 00, P := 1, OUT => #HourString);
       VAL_STRG(IN := #LabelDateTime.MINUTE, SIZE := 2, PREC := 0, FORMAT := 00, P := 1, OUT => #MinuteString);
       VAL_STRG(IN := #LabelDateTime.SECOND, SIZE := 2, PREC := 0, FORMAT := 00, P := 1, OUT => #SecondString);
       #DateTimeString := CONCAT(IN1 := #YearString, IN2 := '/');
       #DateTimeString := CONCAT(IN1 := #DateTimeString, IN2 := #MonthString);
       #DateTimeString := CONCAT(IN1 := #DateTimeString, IN2 := '/');
       #DateTimeString := CONCAT(IN1 := #DateTimeString, IN2 := #DayString);
       #DateTimeString := CONCAT(IN1 := #DateTimeString, IN2 := ' ');
       #DateTimeString := CONCAT(IN1 := #DateTimeString, IN2 := #HourString);
       #DateTimeString := CONCAT(IN1 := #DateTimeString, IN2 := ':');
       #DateTimeString := CONCAT(IN1 := #DateTimeString, IN2 := #MinuteString);
       #DateTimeString := CONCAT(IN1 := #DateTimeString, IN2 := ':');
       #DateTimeString := CONCAT(IN1 := #DateTimeString, IN2 := #SecondString);
   END_IF;
END_REGION

REGION Network 3: Barcode Data Build
   // ENO of a box is taken as its EN; it also drops when the box reports an error
   IF #Print THEN
       VAL_STRG(IN := #SerialNumber, SIZE := 3, PREC := 0, FORMAT := 000, P := 1, OUT => #SerialNumberStringTemp);
       #SerialNumberString := CONCAT(IN1 := #DateTimeString, IN2 := #SerialNumberStringTemp);
       #BarcodeString := CONCAT(IN1 := #PartNumber, IN2 := '|');
       #BarcodeString := CONCAT(IN1 := #BarcodeString, IN2 := #SerialNumberString);
   END_IF;
END_REGION

REGION Network 4
   RUNG wire#powerrail
      Contact( #Print )
      Coil( #Enable )
   END_RUNG
   // the same network as SCL:
   #Enable := #Print;
END_REGION

REGION Network 5: Label Data Build
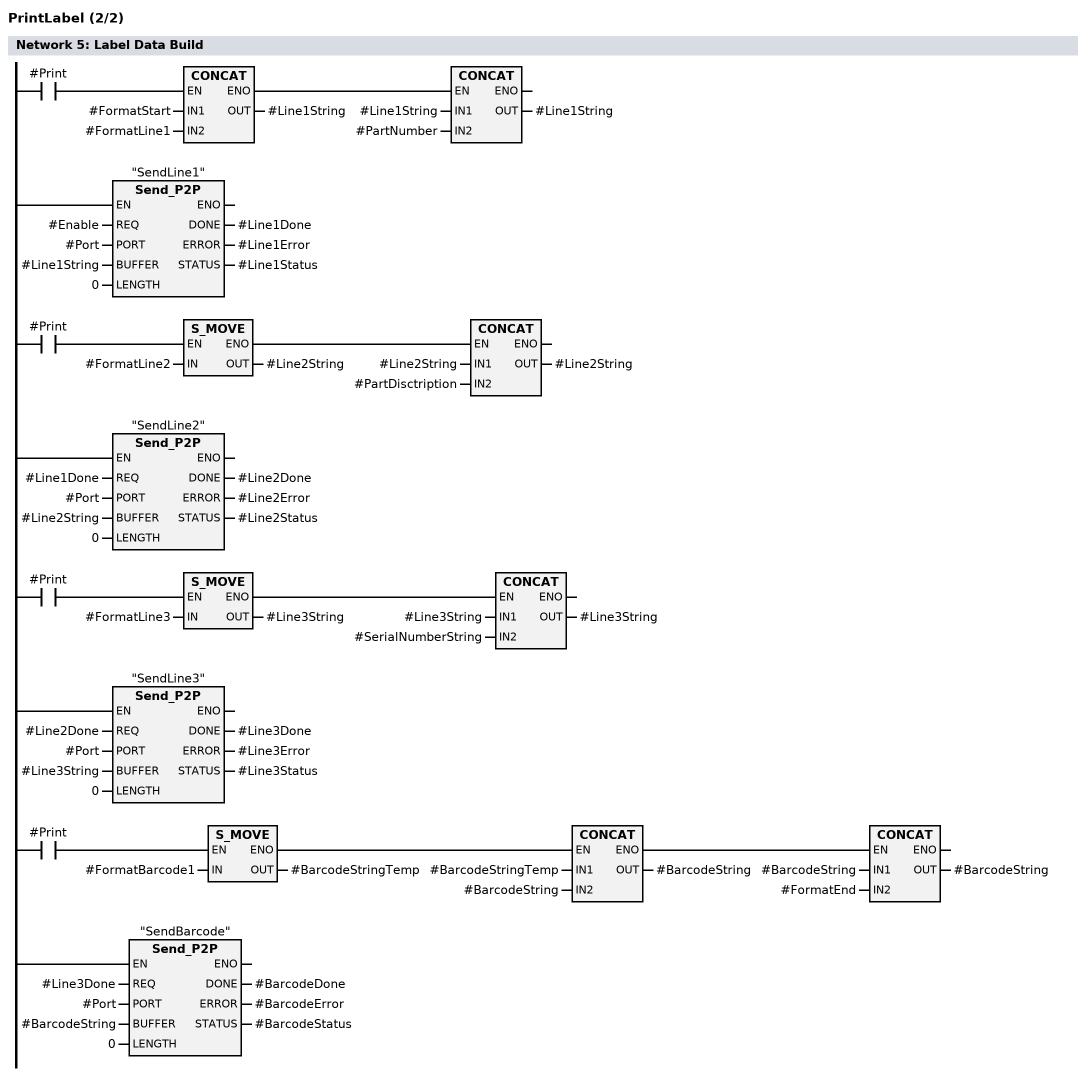
   IF #Print THEN
       #Line1String := CONCAT(IN1 := #FormatStart, IN2 := #FormatLine1);
       #Line1String := CONCAT(IN1 := #Line1String, IN2 := #PartNumber);
   END_IF;
   "SendLine1"(REQ := #Enable,   // Send_P2P
               PORT := #Port,
               BUFFER := #Line1String,
               LENGTH := 0,
               DONE => #Line1Done,
               ERROR => #Line1Error,
               STATUS => #Line1Status);
   IF #Print THEN
       #Line2String := #FormatLine2;
       #Line2String := CONCAT(IN1 := #Line2String, IN2 := #PartDisctription);
   END_IF;
   "SendLine2"(REQ := #Line1Done,   // Send_P2P
               PORT := #Port,
               BUFFER := #Line2String,
               LENGTH := 0,
               DONE => #Line2Done,
               ERROR => #Line2Error,
               STATUS => #Line2Status);
   IF #Print THEN
       #Line3String := #FormatLine3;
       #Line3String := CONCAT(IN1 := #Line3String, IN2 := #SerialNumberString);
   END_IF;
   "SendLine3"(REQ := #Line2Done,   // Send_P2P
               PORT := #Port,
               BUFFER := #Line3String,
               LENGTH := 0,
               DONE => #Line3Done,
               ERROR => #Line3Error,
               STATUS => #Line3Status);
   IF #Print THEN
       #BarcodeStringTemp := #FormatBarcode1;
       #BarcodeString := CONCAT(IN1 := #BarcodeStringTemp, IN2 := #BarcodeString);
       #BarcodeString := CONCAT(IN1 := #BarcodeString, IN2 := #FormatEnd);
   END_IF;
   "SendBarcode"(REQ := #Line3Done,   // Send_P2P
                 PORT := #Port,
                 BUFFER := #BarcodeString,
                 LENGTH := 0,
                 DONE => #BarcodeDone,
                 ERROR => #BarcodeError,
                 STATUS => #BarcodeStatus);
END_REGION
END_FUNCTION_BLOCK